# EPICS StreamDevice protocol: arduinoepics/abacus/abacus.proto
Terminator = CR LF;
replytimeout = 1000;

debug{
    out "%s";
    in "%39c";
}

testled_get{
    out "tled?";
    in "tled:%{0|1}";
}

testled_set{
    out "%{off|on}";
    @init{testled_get;}
}

pled_get{
    out "pled?";
    in "pled:%i";
    @init{ out "pled?"; in "pled:%i"}
}

pled_set{
    out "pled %{0|1}";
    @init{ pled_get; }
}

GetCurr {
    out "meas:curr?";
    in "curr_get:%f";
    @init { out "meas:curr?"; in "curr_get:%f"}
}

GetVolt {
    out "meas:volt?";
    in "volt_get:%f";
    @init { out "meas:volt?"; in "volt_get:%f"}
}

SetVolt {
    out "volt %.4f";
    @init { out "volt?"; in "volt_set:%f" }
    @mismatch{ in "Error: Voltage out of range"; }
}

SetCurr {
    out "curr %.4f";
    @init { out "curr?"; in "curr_set:%f" }
}

GetOutput {
    out "outp?";
    in "outp:%i";
    @init { out "outp?"; in "outp:%i"}
}

SetOutput {
    out "outp %{0|1}";
    @init { GetOutput;}
}
